{attribute addProperty BoxType "EL3783-0000-0018"}
{attribute addProperty Id "High_Current_RangeAT %I*ARRAY [0..3] OF USINT3241High_Current_Range_ActiveAT %I*BOOL815"}
{attribute addProperty CRC "1902850566"}
{attribute addProperty SizeInBites "40"}
{attribute addProperty SizeInBytes "5"}
TYPE AI_Current_Range_716B3206 :
STRUCT
	{attribute addProperty Name "High_Current_Range"}
	High_Current_Range AT %I* : ARRAY [0..3] OF USINT;
	{attribute addProperty Name "High_Current_Range_Active"}
	High_Current_Range_Active AT %I* : BOOL;
END_STRUCT
END_TYPE

(* stored: Version 1.2.0.0, ProductVersion 3.1.4024.9
   DUT AI_Current_Range_716B3206: Id {f7598e7e-ba46-4c30-8ee0-99d406598207} *)
